FUNCTION_BLOCK Utilidades
VAR_INPUT
END_VAR
VAR_OUTPUT
END_VAR
VAR
sJustificaParoComun:STRING;
END_VAR

//Direccionamiento de variables para enviar 
Var_Com_CH2_CH3.aStringCom[62] := Fecha_PLC.StringDateHourMin;

END_FUNCTION_BLOCK

(* stored: Version 1.1.0.1, ProductVersion 3.1.4024.12
   POU Utilidades: Id {63cd07ee-28a3-4f22-aefc-aaddc9ee9d5c}, SpecialFunc None *)
